// Chainable string builder interface.
INTERFACE INTERNAL I_Strb EXTENDS I_Debug

// Appends text; truncates at 255 chars.
METHOD Append : I_Strb
VAR_INPUT
    sToAdd : Str; // Text to append.
END_VAR
END_METHOD

// Finds first match after position; outputs zero positions when not found.
METHOD FindFirstAfter : I_Strb
VAR_INPUT
    sToFind : Str;      // Text to find.
    nPosition : INT := 1; // One-based start position.
END_VAR
VAR_OUTPUT
    nStart : INT;       // Match start, or 0.
    nEnd : INT;         // Match end, or 0.
END_VAR
END_METHOD

// Finds last match before position; outputs zero positions when not found.
METHOD FindLastBefore : I_Strb
VAR_INPUT
    sToFind : Str;        // Text to find.
    nPosition : INT := 256; // One-based end position; 256 means current length.
END_VAR
VAR_OUTPUT
    nStart : INT;         // Match start, or 0.
    nEnd : INT;           // Match end, or 0.
END_VAR
END_METHOD

// Returns current text.
METHOD Get : Str
VAR_INPUT
END_VAR
END_METHOD

// Returns current length.
METHOD GetLength : INT
VAR_INPUT
END_VAR
END_METHOD

// TRUE when text is found after position.
METHOD HasAfter : BOOL
VAR_INPUT
    sToFind : Str;      // Text to find.
    nPosition : INT := 0; // One-based start position.
END_VAR
VAR_OUTPUT
    nStart : INT;       // Match start, or 0.
    nEnd : INT;         // Match end, or 0.
END_VAR
END_METHOD

// TRUE when text is found before position.
METHOD HasBefore : BOOL
VAR_INPUT
    sToFind : Str;        // Text to find.
    nPosition : INT := 256; // One-based end position; 256 means current length.
END_VAR
VAR_OUTPUT
    nStart : INT;         // Match start, or 0.
    nEnd : INT;           // Match end, or 0.
END_VAR
END_METHOD

// Inserts text; no change when position is invalid.
METHOD Inject : I_Strb
VAR_INPUT
    nPosition : INT;    // One-based insert position.
    sToInject : Str;    // Text to insert.
END_VAR
END_METHOD

// TRUE when current length is 0.
METHOD IsEmpty : BOOL
VAR_INPUT
END_VAR
END_METHOD

// Outputs current length and returns this builder.
METHOD Length : I_Strb
VAR_OUTPUT
	nLen: INT; // Current length.
END_VAR
END_METHOD

// Prepends text; truncates at 255 chars.
METHOD Prepend : I_Strb
VAR_INPUT
    sToAdd : Str; // Text to prepend.
END_VAR
END_METHOD

// Removes text; no change when position or length is invalid.
METHOD Remove : I_Strb
VAR_INPUT
    nLength : INT;    // Characters to remove.
    nPosition : INT;  // One-based start position.
END_VAR
END_METHOD

// Sets current text.
METHOD Set : I_Strb
VAR_INPUT
    sValue : Str; // New text.
END_VAR
END_METHOD

// Copies substring into sSlice; no change when position or length is invalid.
METHOD Slice : I_Strb
VAR_INPUT
	nLength : INT;   // Characters to copy.
    nPosition : INT; // One-based start position.
END_VAR
VAR_OUTPUT
    sSlice : Strb;   // Output slice builder.
END_VAR
END_METHOD

// Splits text into left and right builders.
METHOD Split : I_Strb
VAR_INPUT
    nPosition : INT; // One-based split position.
END_VAR
VAR_OUTPUT
    sLeft : Strb;    // Left side.
    sRight : Strb;   // Right side.
END_VAR
END_METHOD

// Outputs current text and returns this builder.
METHOD Write : I_Strb;
VAR_OUTPUT
	sOut: Str; // Current text.
END_VAR
END_METHOD

END_INTERFACE

(* stored: Version 1.1.0.1
   Itf I_Strb: Id {ba21f907-2947-410b-a5fe-d31c0fb60621}
   Method Append: Id {248d4e6a-1d63-4a88-a9ff-6f22af843738}
   Method FindFirstAfter: Id {cbb45280-4d0a-46e0-9518-44d206a10b65}
   Method FindLastBefore: Id {4605251b-2100-457a-9572-22dbfde23e5d}
   Method Get: Id {3e18555f-93c7-4867-826e-d1df008ba5f5}
   Method GetLength: Id {28af4e6d-e908-4012-808f-6bdc656fda8d}
   Method HasAfter: Id {f6606593-96a5-466f-bbd2-567dc49ba5e1}
   Method HasBefore: Id {3ba32025-a527-449a-a307-df9b66ed9eda}
   Method Inject: Id {42b4e730-2675-4489-9fe4-217e8e7d42d0}
   Method IsEmpty: Id {da0eb481-a681-4dc1-a9b6-bcdbbaeca255}
   Method Length: Id {a89198ee-1469-4ece-8be4-81bee1841744}
   Method Prepend: Id {5bc04033-c6a6-47d8-8c78-bbe521b9bc45}
   Method Remove: Id {38c87d18-4637-4049-b384-460f530c2152}
   Method Set: Id {cde054de-26e3-4022-b4ee-a7751f8859aa}
   Method Slice: Id {c5d2cbbd-cd3e-4818-966c-244420d51bcb}
   Method Split: Id {827c2322-1e1a-4752-891a-627fe8cdc2d1}
   Method Write: Id {70df4ad8-01ef-4ed4-8373-85eed225ddfa} *)
